ABB RAPID module: Target_L.mod

MODULE Target_L
    CONST robtarget TG_check_DUL:=[[334.53,153.09,413.36],[0.0231746,-0.0106126,0.706656,-0.707098],[0,0,0,4],[163.271,9E+09,9E+09,9E+09,9E+09,9E+09]];
    CONST robtarget check_DUL:=[[334.59,18.17,413.39],[0.0233478,-0.0105724,0.706721,-0.707028],[-1,0,0,4],[163.279,9E+09,9E+09,9E+09,9E+09,9E+09]];
    CONST robtarget check_L:=[[351.03,-2.57,412.40],[0.464957,-0.506158,-0.497292,0.529452],[-1,0,0,4],[146.859,9E+09,9E+09,9E+09,9E+09,9E+09]];
    CONST robtarget center:=[[319.999933883,19.799690761,200.00026097],[0.000038341,0.000014091,-0.707108747,0.707104814],[-1,0,0,4],[162.87092765,9E+09,9E+09,9E+09,9E+09,9E+09]];
    CONST robtarget home:=[[89.387954366,156.622115869,147.913470331],[0.066010721,0.842420916,-0.111214905,0.523068666],[0,0,0,4],[101.964426493,9E+09,9E+09,9E+09,9E+09,9E+09]];
    CONST robtarget TG_case_2:=[[319.994696463,80.183849872,200.005143308],[0.500025811,0.500011388,-0.499991422,0.499971378],[-1,0,0,4],[162.870928858,9E+09,9E+09,9E+09,9E+09,9E+09]];
    CONST robtarget TG_case_4:=[[319.994807344,80.184031378,200.005043033],[0.499971262,0.499991405,0.50001148,-0.500025851],[-1,0,1,4],[162.870927234,9E+09,9E+09,9E+09,9E+09,9E+09]];
    CONST robtarget TG_case_5:=[[300,-0.2,200],[0,0.707106781,0,0.707106781],[-1,0,0,4],[162.870927482,9E+09,9E+09,9E+09,9E+09,9E+09]];
    CONST robtarget TG_case_5_1:=[[250.000099956,-0.199840787,199.999926771],[-0.000000024,0.707106903,-0.000000114,0.707106659],[-1,-1,1,4],[162.870928855,9E+09,9E+09,9E+09,9E+09,9E+09]];
    CONST robtarget TG_case_5_2:=[[250.000197537,149.80033722,199.999844719],[0.000000025,0.707107009,-0.000000212,0.707106554],[-1,-1,1,4],[162.870925691,9E+09,9E+09,9E+09,9E+09,9E+09]];
    CONST robtarget TG_case_6:=[[300.000082163,-0.199866648,199.999889141],[0.499999899,-0.50000005,0.500000191,-0.49999986],[-1,-1,1,4],[162.870919843,9E+09,9E+09,9E+09,9E+09,9E+09]];
    CONST robtarget TG_case_6_1:=[[250.000175623,-0.199692427,199.999819226],[0.499999803,-0.500000087,0.500000347,-0.499999762],[-1,-1,2,4],[162.870928131,9E+09,9E+09,9E+09,9E+09,9E+09]];
    CONST robtarget TG_case_6_2:=[[250.000293205,149.800491851,199.999729037],[0.499999707,-0.500000069,0.500000576,-0.499999648],[-1,-1,2,4],[162.87093138,9E+09,9E+09,9E+09,9E+09,9E+09]];
    CONST robtarget TG_case_8:=[[319.994696463,70.183849872,200.005143308],[0.707104794,0.707108768,0.000014118,-0.00003849],[-1,0,-2,4],[162.870928858,9E+09,9E+09,9E+09,9E+09,9E+09]];
    CONST robtarget TG_case_9:=[[320.000214982,-0.199651003,269.999812927],[0.000000178,1,-0.000000116,-0.00000022],[-1,1,1,4],[161.217311934,9E+09,9E+09,9E+09,9E+09,9E+09]];
    CONST robtarget TG_case_9_1:=[[320.000307354,99.800522072,269.999705455],[0.000000306,1,-0.00000018,-0.000000393],[-1,1,1,4],[161.217317735,9E+09,9E+09,9E+09,9E+09,9E+09]];
    CONST robtarget TG_case_10:=[[320,-0.2,220],[0,-0.707106781,0.707106781,0],[-1,1,2,4],[162.870926162,9E+09,9E+09,9E+09,9E+09,9E+09]];
    CONST robtarget TG_case_10_1:=[[320.000079696,-0.199814515,269.999909403],[-0.000000053,-0.70710675,0.707106812,0.000000216],[-1,1,2,4],[162.870931791,9E+09,9E+09,9E+09,9E+09,9E+09]];
    CONST robtarget TG_case_10_2:=[[320.000209695,99.800354027,269.99981139],[-0.000000079,-0.707106755,0.707106807,0.000000394],[-1,1,2,4],[162.870927719,9E+09,9E+09,9E+09,9E+09,9E+09]];
    CONST robtarget TG_case_11_1:=[[320.000098301,-0.199812602,269.999917664],[-0.000000089,0.000000062,1,0.000000114],[-1,1,-1,4],[161.217313884,9E+09,9E+09,9E+09,9E+09,9E+09]];
    CONST robtarget TG_case_11_2:=[[320.000224741,99.800346333,269.999826105],[-0.000000185,0.000000151,1,0.000000196],[-1,1,-1,4],[161.217312013,9E+09,9E+09,9E+09,9E+09,9E+09]];
    CONST robtarget TG_case_12:=[[320.000098301,-0.199812602,219.999917664],[0.000000144,0.707106825,0.707106737,0.000000018],[-1,1,-1,4],[161.217313884,9E+09,9E+09,9E+09,9E+09,9E+09]];
    CONST robtarget TG_case_12_1:=[[320.000215513,-0.199633112,269.999809709],[0.000000322,0.707106887,0.707106676,0.000000014],[-1,1,0,4],[161.217312281,9E+09,9E+09,9E+09,9E+09,9E+09]];
    CONST robtarget TG_case_12_2:=[[320.000215513,99.800366888,269.999809709],[-0.000000322,0.707106887,0.707106676,0.000000014],[-1,1,0,4],[161.217312281,9E+09,9E+09,9E+09,9E+09,9E+09]];
    CONST robtarget TG_case_19_1:=[[320.000098301,-0.199812602,269.999917664],[-0.000000089,0.000000062,1,0.000000114],[-1,1,-1,4],[161.217313884,9E+09,9E+09,9E+09,9E+09,9E+09]];
    CONST robtarget TG_case_19_2:=[[320.000224741,99.800346333,269.999826105],[-0.000000185,0.000000151,1,0.000000196],[-1,1,-1,4],[161.217312013,9E+09,9E+09,9E+09,9E+09,9E+09]];
    CONST robtarget TG_case_21:=[[319.994696463,70.183849872,200.005143308],[0.707104794,0.707108768,0.000014118,-0.00003849],[-1,0,-2,4],[162.870928858,9E+09,9E+09,9E+09,9E+09,9E+09]];
    CONST robtarget waitpoint:=[[319.994777109,110.184043671,200.005015932],[0.00003863,0.00001422,-0.707108856,0.707104705],[-1,0,0,4],[162.870926162,9E+09,9E+09,9E+09,9E+09,9E+09]];
    CONST robtarget rotate_BFR:=[[320.000426173,34.800029407,199.999961671],[0.000038637,0.00001417,-0.707108854,0.707104707],[-1,0,0,4],[162.870928931,9E+09,9E+09,9E+09,9E+09,9E+09]];
    CONST robtarget TG_rotate_x2:=[[319.994968105,80.184371446,200.004837009],[0.707104525,0.707109036,0.000014283,-0.000038978],[-1,0,-2,4],[162.87093396,9E+09,9E+09,9E+09,9E+09,9E+09]];
    CONST robtarget rotate_D:=[[320.000098301,-0.199812602,219.999917664],[0.000000114,1,-0.000000062,-0.000000089],[-1,1,1,4],[161.217313884,9E+09,9E+09,9E+09,9E+09,9E+09]];
    CONST robtarget rotate_U:=[[320,-0.2,220],[0,0,1,0],[-1,1,-1,4],[161.217313243,9E+09,9E+09,9E+09,9E+09,9E+09]];
    CONST robtarget TG_rotate_CCW:=[[319.99500521,80.055194631,200.004835821],[0.500025916,0.500011691,-0.499991481,0.49997091],[-1,0,0,4],[162.870927681,9E+09,9E+09,9E+09,9E+09,9E+09]];
    CONST robtarget TG_rotate_CW:=[[319.994916659,80.055008682,200.004912248],[0.499971026,0.499991503,0.500011628,-0.500025842],[-1,0,0,4],[162.870929188,9E+09,9E+09,9E+09,9E+09,9E+09]];
ENDMODULE
